// TIA Portal project "Mezcla_Dos_Liquidos" (V16)

(* hardware
DEVICE "S71500/ET200MP station_1"  S7-1500 station
   slot 0: "Perfil soporte_0"  Rack  6ES7 590-1***0-0AA0
   slot 1: "PLC_1"  CPU 1512C-1 PN  6ES7 512-1CK00-0AB0  V2.8
      slot 3: "Display de la CPU_1"  6ES7591-1AA00-0AA0
      slot 32768: "Interfaz PROFINET_1"  X1
         slot 32769: "Puerto_1"  X1 P1
         slot 32770: "Puerto_2"  X1 P2
      slot 34817: "Virtual CP interface port_1"  Virtual CP interface port  Virtual CP interface port
*)

// ===== PLC "PLC_1"  CPU 1512C-1 PN =====

VAR_GLOBAL   // PLC tag table "Entradas"
   "Marcha" AT %I4.0 : Bool;
   "Paro" AT %I4.1 : Bool;
   "PSeleccion" AT %I4.2 : Bool;
   "s0" AT %I5.0 : Bool;
   "s1" AT %I5.1 : Bool;
   "s2" AT %I5.2 : Bool;
   "s3" AT %I5.3 : Bool;
   "s4" AT %I5.4 : Bool;
   "s5" AT %I5.5 : Bool;
END_VAR

VAR_GLOBAL   // PLC tag table "Salidas"
   "EV_liquidoA" AT %Q0.0 : Bool;
   "EV_liquidoB" AT %Q0.1 : Bool;
   "EV_Vaciado" AT %Q0.2 : Bool;
   "Agitador" AT %Q0.3 : Bool;
   "EV_Desecho" AT %Q0.4 : Bool;
END_VAR

VAR_GLOBAL   // PLC tag table "Señales_de_Control"
   "Inicio" AT %M0.0 : Bool;
   "SolCondIni" AT %M0.1 : Bool;
   "FinCondIni" AT %M0.2 : Bool;
   "ProdNormal" AT %M0.3 : Bool;
   "ParoFC" AT %M0.4 : Bool;
   "FinProceso" AT %M0.5 : Bool;
   "SolMarcha" AT %M0.6 : Bool;
   "FinMarchaFin" AT %M0.7 : Bool;
   "Marcha_AUX" AT %M10.0 : Bool;
   "Marcha_FA" AT %M10.1 : Bool;
   "Paro_AUX" AT %M11.0 : Bool;
   "Paro_FA" AT %M11.1 : Bool;
END_VAR

DATA_BLOCK "SecPrincipal_DB"   // DB1
{ S7_Optimized_Access := 'TRUE' }
VERSION : 0.1
// stored: InstanceOfName SecPrincipal
"SecPrincipal"
BEGIN
END_DATA_BLOCK

// folder: System blocks/Program resources

DATA_BLOCK "Cont_DB"   // DB2
{ S7_Optimized_Access := 'TRUE' }
AUTHOR : Simatic
FAMILY : IEC
NAME : CNTR
VERSION : 1.0
// stored: InstanceOfName IEC_COUNTER
"IEC_COUNTER"
BEGIN
END_DATA_BLOCK

// folder: (top level)

FUNCTION_BLOCK "SecPrincipal"   // FB1, GRAPH_PLUS
{ S7_Optimized_Access := 'TRUE' }
VERSION : 0.1
   VAR_INPUT
      OFF_SQ : Bool := false;   // Desactivar cadena
      INIT_SQ : Bool := false;   // Poner cadena en estado inicial
      ACK_EF : Bool := false;   // Acusar todos los errores y fallos
      S_PREV : Bool := false;   // Mostrar la etapa anterior en el parámetro S_NO
      S_NEXT : Bool := false;   // Mostrar la etapa siguiente en el parámetro S_NO
      SW_AUTO : Bool := false;   // Modo automático
      SW_TAP : Bool := false;   // Semiautomático/continuar con transición
      SW_TOP : Bool := false;   // Semiautomático/transición ignorada
      SW_MAN : Bool := false;   // Modo manual
      S_SEL : Int := 0;   // Seleccionar la etapa que debe mostrarse en S_NO
      S_ON : Bool := false;   // Activar la etapa del parámetro S_NO
      S_OFF : Bool := false;   // Desactivar el incremento presente en el parámetro S_NO
      T_PUSH : Bool := false;   // Habilitar conmutación de transición en modo semiautomático
   END_VAR
   VAR_OUTPUT
      S_NO : Int := 0;   // Número de etapa
      S_MORE : Bool := false;   // Existen más etapas que pueden mostrarse en S_NO.
      S_ACTIVE : Bool := false;   // El incremento presente en el parámetro S_NO está activo
      ERR_FLT : Bool := false;   // Error de grupo interlock o supervisión
      AUTO_ON : Bool := false;   // Modo automático activado
      TAP_ON : Bool := false;   // Modo semiautomático/etapa con transición activada
      TOP_ON : Bool := false;   // Modo semiautomático/Ignorar transición activado
      MAN_ON : Bool := false;   // Modo manual activado
   END_VAR
   VAR
      HMI_INFO : Array[0..0] of UInt;
      RT_DATA : G7_RTDataPlus_V6;   // Área de datos interna
      Trans1 : G7_TransitionPlus_V6;   // Estructura de la transición
      X0 : G7_StepPlus_V6;   // Estructura de la etapa
      X1 : G7_StepPlus_V6;   // Estructura de la etapa
      Trans2 : G7_TransitionPlus_V6;   // Estructura de la transición
      X2 : G7_StepPlus_V6;   // Estructura de la etapa
      Trans3 : G7_TransitionPlus_V6;   // Estructura de la transición
      X3 : G7_StepPlus_V6;   // Estructura de la etapa
      Trans4 : G7_TransitionPlus_V6;   // Estructura de la transición
      X4 : G7_StepPlus_V6;   // Estructura de la etapa
      Trans5 : G7_TransitionPlus_V6;   // Estructura de la transición
   END_VAR
BEGIN
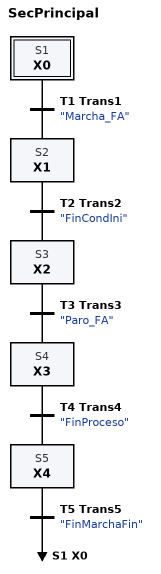
   // sequencer 1
   INITIAL_STEP X0:   // S1, max time T#10S, warning time T#7S
   END_STEP
   TRANSITION Trans1 FROM X0 TO X1   // T1
      := "Marcha_FA";
   END_TRANSITION
   STEP X1:   // S2, max time T#10S, warning time T#7S
   END_STEP
   TRANSITION Trans2 FROM X1 TO X2   // T2
      := "FinCondIni";
   END_TRANSITION
   STEP X2:   // S3, max time T#10S, warning time T#7S
   END_STEP
   TRANSITION Trans3 FROM X2 TO X3   // T3
      := "Paro_FA";
   END_TRANSITION
   STEP X3:   // S4, max time T#10S, warning time T#7S
   END_STEP
   TRANSITION Trans4 FROM X3 TO X4   // T4
      := "FinProceso";
   END_TRANSITION
   STEP X4:   // S5, max time T#10S, warning time T#7S
   END_STEP
   TRANSITION Trans5 FROM X4 TO X0   // T5, jump
      := "FinMarchaFin";
   END_TRANSITION
END_FUNCTION_BLOCK

FUNCTION_BLOCK "CondIni"   // FB2, GRAPH_PLUS
{ S7_Optimized_Access := 'TRUE' }
VERSION : 0.1
   VAR_INPUT
      OFF_SQ : Bool := false;   // Desactivar cadena
      INIT_SQ : Bool := false;   // Poner cadena en estado inicial
      ACK_EF : Bool := false;   // Acusar todos los errores y fallos
      S_PREV : Bool := false;   // Mostrar la etapa anterior en el parámetro S_NO
      S_NEXT : Bool := false;   // Mostrar la etapa siguiente en el parámetro S_NO
      SW_AUTO : Bool := false;   // Modo automático
      SW_TAP : Bool := false;   // Semiautomático/continuar con transición
      SW_TOP : Bool := false;   // Semiautomático/transición ignorada
      SW_MAN : Bool := false;   // Modo manual
      S_SEL : Int := 0;   // Seleccionar la etapa que debe mostrarse en S_NO
      S_ON : Bool := false;   // Activar la etapa del parámetro S_NO
      S_OFF : Bool := false;   // Desactivar el incremento presente en el parámetro S_NO
      T_PUSH : Bool := false;   // Habilitar conmutación de transición en modo semiautomático
   END_VAR
   VAR_OUTPUT
      S_NO : Int := 0;   // Número de etapa
      S_MORE : Bool := false;   // Existen más etapas que pueden mostrarse en S_NO.
      S_ACTIVE : Bool := false;   // El incremento presente en el parámetro S_NO está activo
      ERR_FLT : Bool := false;   // Error de grupo interlock o supervisión
      AUTO_ON : Bool := false;   // Modo automático activado
      TAP_ON : Bool := false;   // Modo semiautomático/etapa con transición activada
      TOP_ON : Bool := false;   // Modo semiautomático/Ignorar transición activado
      MAN_ON : Bool := false;   // Modo manual activado
   END_VAR
   VAR
      HMI_INFO : Array[0..0] of UInt;
      RT_DATA : G7_RTDataPlus_V6;   // Área de datos interna
      Trans1 : G7_TransitionPlus_V6;   // Estructura de la transición
      Step1 : G7_StepPlus_V6;   // Estructura de la etapa
   END_VAR
BEGIN
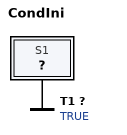
   // sequencer 1
   INITIAL_STEP "?":   // S1
   END_STEP
   TRANSITION "?" FROM "?" TO ?   // T1
      := TRUE;
   END_TRANSITION
END_FUNCTION_BLOCK

FUNCTION_BLOCK "MarchaFin"   // FB3, GRAPH_PLUS
{ S7_Optimized_Access := 'TRUE' }
VERSION : 0.1
   VAR_INPUT
      OFF_SQ : Bool := false;   // Desactivar cadena
      INIT_SQ : Bool := false;   // Poner cadena en estado inicial
      ACK_EF : Bool := false;   // Acusar todos los errores y fallos
      S_PREV : Bool := false;   // Mostrar la etapa anterior en el parámetro S_NO
      S_NEXT : Bool := false;   // Mostrar la etapa siguiente en el parámetro S_NO
      SW_AUTO : Bool := false;   // Modo automático
      SW_TAP : Bool := false;   // Semiautomático/continuar con transición
      SW_TOP : Bool := false;   // Semiautomático/transición ignorada
      SW_MAN : Bool := false;   // Modo manual
      S_SEL : Int := 0;   // Seleccionar la etapa que debe mostrarse en S_NO
      S_ON : Bool := false;   // Activar la etapa del parámetro S_NO
      S_OFF : Bool := false;   // Desactivar el incremento presente en el parámetro S_NO
      T_PUSH : Bool := false;   // Habilitar conmutación de transición en modo semiautomático
   END_VAR
   VAR_OUTPUT
      S_NO : Int := 0;   // Número de etapa
      S_MORE : Bool := false;   // Existen más etapas que pueden mostrarse en S_NO.
      S_ACTIVE : Bool := false;   // El incremento presente en el parámetro S_NO está activo
      ERR_FLT : Bool := false;   // Error de grupo interlock o supervisión
      AUTO_ON : Bool := false;   // Modo automático activado
      TAP_ON : Bool := false;   // Modo semiautomático/etapa con transición activada
      TOP_ON : Bool := false;   // Modo semiautomático/Ignorar transición activado
      MAN_ON : Bool := false;   // Modo manual activado
   END_VAR
   VAR
      HMI_INFO : Array[0..0] of UInt;
      RT_DATA : G7_RTDataPlus_V6;   // Área de datos interna
      Trans1 : G7_TransitionPlus_V6;   // Estructura de la transición
      X70 : G7_StepPlus_V6;   // Estructura de la etapa
      X71 : G7_StepPlus_V6;   // Estructura de la etapa
      Trans2 : G7_TransitionPlus_V6;   // Estructura de la transición
      X72 : G7_StepPlus_V6;   // Estructura de la etapa
      Trans3 : G7_TransitionPlus_V6;   // Estructura de la transición
   END_VAR
BEGIN
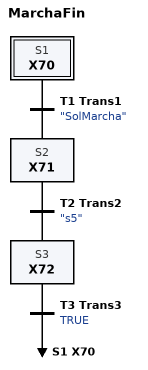
   // sequencer 1
   INITIAL_STEP X70:   // S1, max time T#10S, warning time T#7S
   END_STEP
   TRANSITION Trans1 FROM X70 TO X71   // T1
      := "SolMarcha";
   END_TRANSITION
   STEP X71:   // S2, max time T#10S, warning time T#7S
   END_STEP
   TRANSITION Trans2 FROM X71 TO X72   // T2
      := "s5";
   END_TRANSITION
   STEP X72:   // S3, max time T#10S, warning time T#7S
   END_STEP
   TRANSITION Trans3 FROM X72 TO X70   // T3, jump
      := TRUE;
   END_TRANSITION
END_FUNCTION_BLOCK

ORGANIZATION_BLOCK "Main"   // OB1, LAD, ProgramCycle
TITLE = "Main Program Sweep (Cycle)"
{ S7_Optimized_Access := 'TRUE' }
VERSION : 0.1
   VAR_INPUT
      Initial_Call : Bool;   // Initial call of this OB
      Remanence : Bool;   // =True, if remanent data are available
   END_VAR
   VAR_TEMP   // added for the SCL form of the ladder/FBD networks
      _w1 : Bool;
      _w2 : Bool;
   END_VAR
BEGIN

REGION Network 1: Flancos, Contadores y Temporizadores
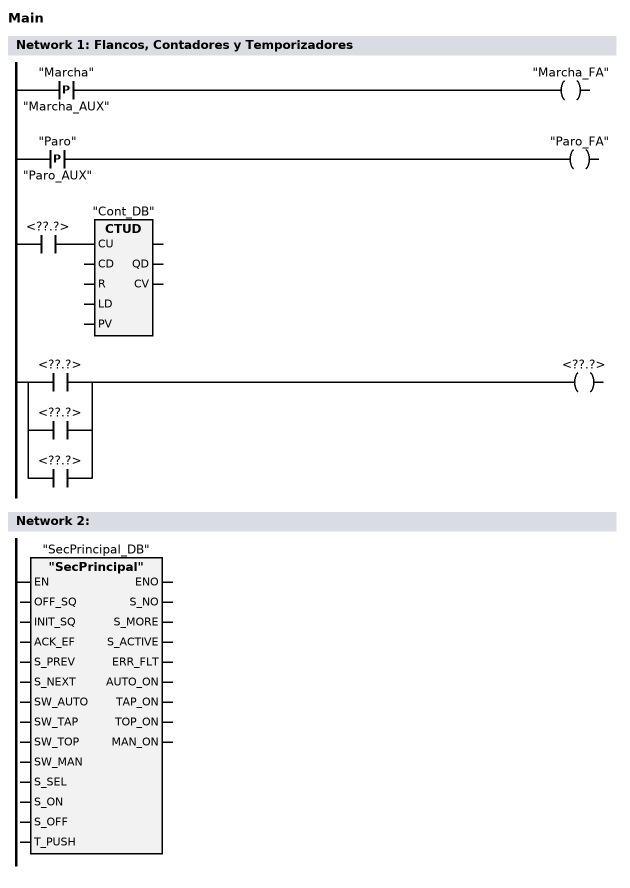
   // no checked SCL form for this network; see the picture
END_REGION

REGION Network 2
   RUNG wire#powerrail
      "SecPrincipal_DB"(OFF_SQ :=, INIT_SQ :=, ACK_EF :=, S_PREV :=, S_NEXT :=, SW_AUTO :=, SW_TAP :=, SW_TOP :=, SW_MAN :=, S_SEL :=, S_ON :=, S_OFF :=, T_PUSH :=, S_NO =>, S_MORE =>, S_ACTIVE =>, ERR_FLT =>, AUTO_ON =>, TAP_ON =>, TOP_ON =>, MAN_ON =>)
   END_RUNG
   // the same network as SCL:
   "SecPrincipal_DB"();   // "SecPrincipal"
END_REGION
END_ORGANIZATION_BLOCK